Fanuc KAREL source: kd00007.KL

-- PROVISIONAL review KL for V1013-1; original PC SHA256 69bb7a041ea7fa94a5ad1490365365f888501cb96fd74553a7fa03d71a495c96
-- Incomplete behavior may be omitted. Consult companion uncertainty JSON. Do not deploy.
PROGRAM KD00007
%NOLOCKGROUP
-- UNRESOLVED_DECL I type=020010
-- UNRESOLVED_DECL J type=020010
-- UNRESOLVED_DECL B type=020012
-- UNRESOLVED_DECL R type=020011
-- UNRESOLVED_DECL S type=021f50
BEGIN
  -- UNRESOLVED_PC offsets 5-12; opcodes 9D,23
  -- UNRESOLVED_PC offsets 17-21; opcodes 7F
END KD00007
